// TwinCAT 3 PLC project Untitled2
// ProgramVersion: 3.1.4023.0
// libraries:
//   Tc2_Standard, * (Beckhoff Automation GmbH)
//   Tc2_System, * (Beckhoff Automation GmbH)
//   Tc3_Module, * (Beckhoff Automation GmbH)
// project tree:
//   / PlcTask.TcTTO
//   POUs/ FB_DisplacementSensor.TcPOU, FB_Test.TcPOU, MAIN.TcPOU
// real-time tasks:
//   TASK PlcTask: cycle T#10ms, priority 20, ADS port 350

CONFIGURATION Untitled2
    RESOURCE PLC ON TwinCAT3
        TASK PlcTask(INTERVAL := T#10ms, PRIORITY := 20);
        PROGRAM MAIN WITH PlcTask : MAIN;
    END_RESOURCE
END_CONFIGURATION

// ---- POUs/MAIN.TcPOU
PROGRAM MAIN
VAR
	fbDispSens : FB_DisplacementSensor();
	fbTest : FBtest();
END_VAR

END_PROGRAM

// ---- POUs/FB_DisplacementSensor.TcPOU
FUNCTION_BLOCK FB_DisplacementSensor

VAR_OUTPUT
	nDistance : INT;
	bInValueRange : BOOL;
END_VAR
VAR
	aInputBytes AT %I* : ARRAY[1..2] OF BYTE;
	nWord1 : WORD;
	nWord2 : WORD;
	nWord3 : WORD;
                                                                                                                                                                                                                                                                                                                                                                                                                                                                                                                                                                                                                                                                                                                                                                                                                                                                                                                                                                                                                                                                                                                                                                                                                                                                                                         I* : ARRAY 
END_VAR

nWord1 := TO_WORD(aInputBytes[1]);

//1111_1111
//0000_0000_1111_1111


nWord2 := aInputBytes[2];
//1111_1111
//0000_0000_1111_1111

nWord1 := SHL(nWord1, 8);
// 1111_1111_0000_0000
nWord3 := nWord1 OR nWord2;
//1111_1111_1111_1111
nWord3 := SHR(nWord3,4);

nDistance := TO_INT(nWord3); 

bInValueRange := aInputBytes[2].0;

END_FUNCTION_BLOCK

// ---- POUs/FB_Test.TcPOU
FUNCTION_BLOCK FB_Test
VAR
	nCounters : LINT;
END_VAR

nCounter := nCounter + 1;

END_FUNCTION_BLOCK
